% RSLogix 500 project PROC1_SCP.RSS, saved by version 8.30.00.16 %
PROJECT "PROC1"    % processor: Bul.1763 MicroLogix 1100 Series B %

PROGRAM FILES
  LAD 2   3 rungs

DATA FILES
  O0 OUTPUT  4 elements
  I1 INPUT  6 elements
  S2 STATUS  66 elements
  B3 BINARY  1 elements
  T4 TIMER  1 elements
  C5 COUNTER  1 elements
  R6 CONTROL  1 elements
  N7 INTEGER  11 elements
  F8 FLOAT  1 elements

LADDER 2
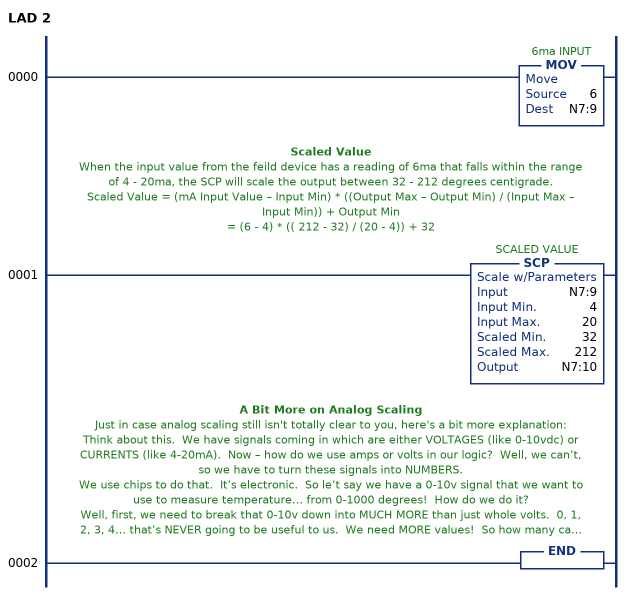
% Rung: 0 %
SOR MOV 6 N7:9 EOR
%   N7:9  "6ma INPUT" %
% Rung: 1 %
% TITLE: Scaled Value %
% When the input value from the feild device has a reading of 6ma that falls within the range of 4 - 20ma, the SCP will scale the output between 32 - 212 degrees centigrade.
% 
% Scaled Value = (mA Input Value – Input Min) * ((Output Max – Output Min) / (Input Max – Input Min)) + Output Min
% 
% 			= (6 - 4) * (( 212 - 32) / (20 - 4)) + 32 %
SOR SCP N7:9 4 20 32 212 N7:10 EOR
%   N7:9  "6ma INPUT" %
%   N7:10  "SCALED VALUE" %
% Rung: 2 %
% TITLE: A Bit More on Analog Scaling %
% Just in case analog scaling still isn't totally clear to you, here's a bit more explanation:
% 
% Think about this.  We have signals coming in which are either VOLTAGES (like 0-10vdc) or CURRENTS (like 4-20mA).  Now – how do we use amps or volts in our logic?  Well, we can’t, so we have to turn these signals into NUMBERS.
% 
% We use chips to do that.  It’s electronic.  So le’t say we have a 0-10v signal that we want to use to measure temperature… from 0-1000 degrees!  How do we do it?
% 
% Well, first, we need to break that 0-10v down into MUCH MORE than just whole volts.  0, 1, 2, 3, 4… that’s NEVER going to be useful to us.  We need MORE values!  So how many can we get?  Well, that depends on our chips (built into our analog IO modules).
% 
% In our case, we have “14-bit” ADC (Analog Digital Converter) chips.  And if we raise 2 to the 14th power, that’ll tell us how many levels of “resolution” we can get out of these chips.  In our case, that number is 16,384.
% 
% So where are we?  We have a temperature sensor capable of reading from 0 to 1000 degrees.  It produces a 0-10v signal.  Our analog input module will convert that signal into a (PID) value – a NUMBER somewhere between 0-16,383, and THAT is what we’ll use in our program!
% 
% But now, we have to turn this number into a temperature value.  When I tell you that the sensor value is 8182, that is MEANINGLESS to you.  You want to know how hot the oven is, right?  So we need to mathematically translate the 0-16,383 value into a temperature value along the range of our sensor’s capability (0-1000 degrees).
% 
% So a sensor value of 0 would represent 0 degrees.
% 
% So a sensor value of 8192 would represent 500 degrees.
% 
% So a sensor value of 16383 would represent 1000 degrees.
% 
% And to calculate that, we can either use a mathematical operation, or simply employ the SCP block which does all the math for us.  So we feed it the address of the input signal, the input range, the output range and finally the destination where we want to store the value.
% 
% 
% 
% Here's a breakdown of how the scaling actually works when an SCP converts a value from one range to another:
% 
% Scaled Value = (mA Input Value – Input Min) * ((Output Max – Output Min) / (Input Max – Input Min)) + Output Min
% 
% where
% 
% mA Input Value = milliamps coming into sensor
% 
% Input Min = minimum value of milliamps coming in
% 
% Input Max = maximum value of milliamps coming in
% 
% Output Min = value represented by Input Min
% 
% Output Max = value represented by Input Max
% 
% 
% 
% So if we had a 4-20mA signal which represented 0-60psi in a tank, and we wanted to see what pressure 9.5mA represents, this is how we would set that up:
% 
% mA Input Value = 9.5
% 
% Input Min = 4
% 
% Input Max = 20
% 
% Output Min = 0
% 
% Output Max = 60
% 
% (9.5 – 4) * ((60 – 0) / (20 – 4)) + 0 = 20.625psi
% 
% 
% 
% If we were scaling a PID value into a temperature range, it would be the same thing.  Suppose we wanted to scale 12250 from PID (0-16383) to a temperature range of 32 to 166 degrees.
% 
% PID Input Value = 12250
% 
% Input Min = 0
% 
% Input Max = 16383
% 
% Output Min = 32
% 
% Output Max = 166
% 
% (12250 – 0) * ((166 – 32) / (16383 – 0)) + 32 = 132.20 degrees %
SOR END EOR

REVISION NOTES
  0: Added comments to rungs

DATA TABLE (non-zero values as saved)
DATA N7
% N7:0 % 0 0 0 0 0 0 0 0 0 6
% N7:10 % 55
